// Mitsubishi GX Works2 project: RecipeMixer2   PLC: FX3U/FX3UC

PROGRAM MAIN
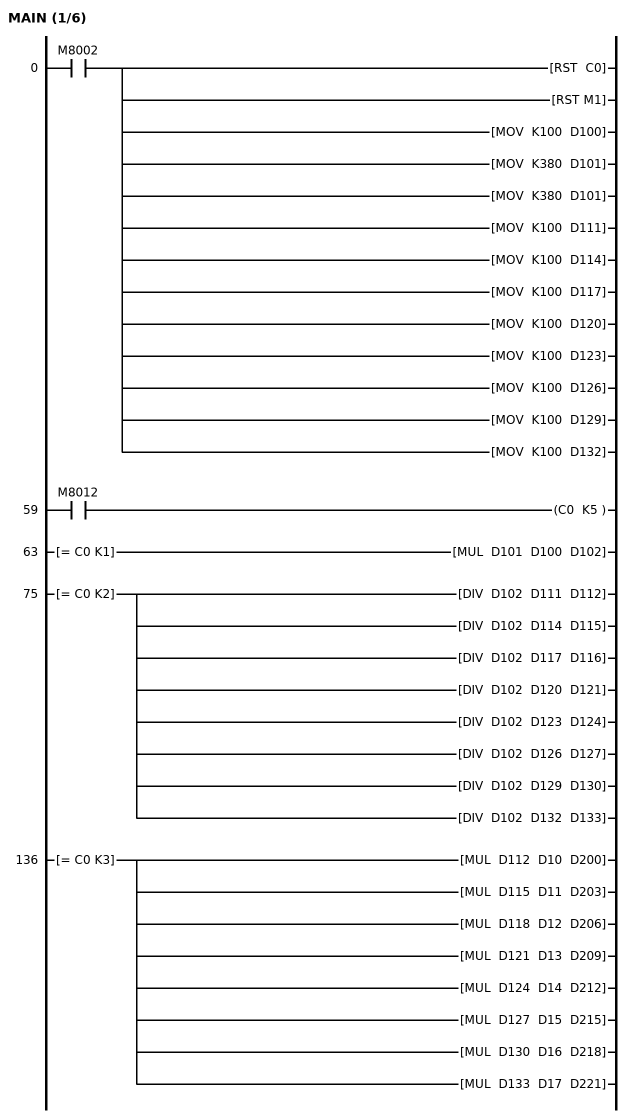
0     LD      M8002
      RST     C0
      RST     M1
      MOV     K100 D100
      MOV     K380 D101
      MOV     K380 D101
      MOV     K100 D111
      MOV     K100 D114
      MOV     K100 D117
      MOV     K100 D120
      MOV     K100 D123
      MOV     K100 D126
      MOV     K100 D129
      MOV     K100 D132
59    LD      M8012
      OUT     C0 K5
63    LD=     C0 K1
      MUL     D101 D100 D102
75    LD=     C0 K2
      DIV     D102 D111 D112
      DIV     D102 D114 D115
      DIV     D102 D117 D116
      DIV     D102 D120 D121
      DIV     D102 D123 D124
      DIV     D102 D126 D127
      DIV     D102 D129 D130
      DIV     D102 D132 D133
136   LD=     C0 K3
      MUL     D112 D10 D200
      MUL     D115 D11 D203
      MUL     D118 D12 D206
      MUL     D121 D13 D209
      MUL     D124 D14 D212
      MUL     D127 D15 D215
      MUL     D130 D16 D218
      MUL     D133 D17 D221
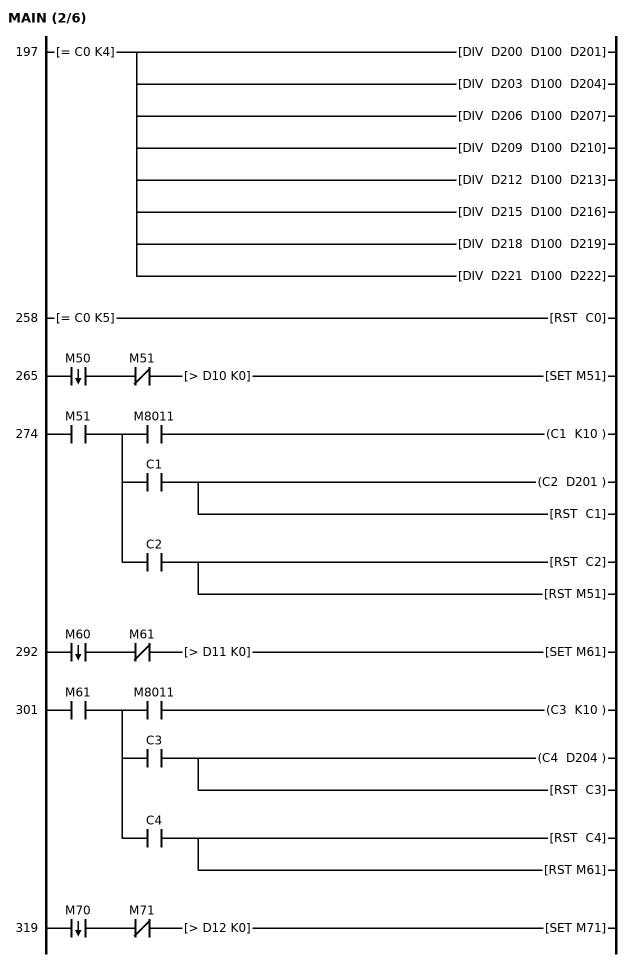
197   LD=     C0 K4
      DIV     D200 D100 D201
      DIV     D203 D100 D204
      DIV     D206 D100 D207
      DIV     D209 D100 D210
      DIV     D212 D100 D213
      DIV     D215 D100 D216
      DIV     D218 D100 D219
      DIV     D221 D100 D222
258   LD=     C0 K5
      RST     C0
265   LDF     M50
      ANI     M51
      AND>    D10 K0
      SET     M51
274   LD      M51
      MPS
      AND     M8011
      OUT     C1 K10
      MRD
      AND     C1
      OUT     C2 D201
      RST     C1
      MPP
      AND     C2
      RST     C2
      RST     M51
292   LDF     M60
      ANI     M61
      AND>    D11 K0
      SET     M61
301   LD      M61
      MPS
      AND     M8011
      OUT     C3 K10
      MRD
      AND     C3
      OUT     C4 D204
      RST     C3
      MPP
      AND     C4
      RST     C4
      RST     M61
319   LDF     M70
      ANI     M71
      AND>    D12 K0
      SET     M71
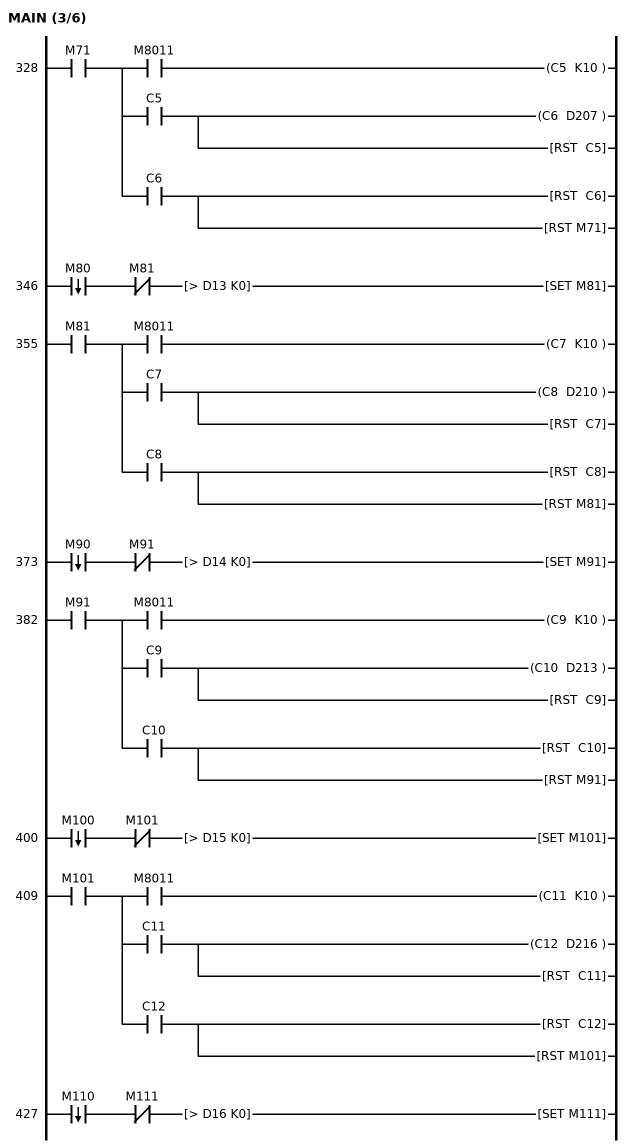
328   LD      M71
      MPS
      AND     M8011
      OUT     C5 K10
      MRD
      AND     C5
      OUT     C6 D207
      RST     C5
      MPP
      AND     C6
      RST     C6
      RST     M71
346   LDF     M80
      ANI     M81
      AND>    D13 K0
      SET     M81
355   LD      M81
      MPS
      AND     M8011
      OUT     C7 K10
      MRD
      AND     C7
      OUT     C8 D210
      RST     C7
      MPP
      AND     C8
      RST     C8
      RST     M81
373   LDF     M90
      ANI     M91
      AND>    D14 K0
      SET     M91
382   LD      M91
      MPS
      AND     M8011
      OUT     C9 K10
      MRD
      AND     C9
      OUT     C10 D213
      RST     C9
      MPP
      AND     C10
      RST     C10
      RST     M91
400   LDF     M100
      ANI     M101
      AND>    D15 K0
      SET     M101
409   LD      M101
      MPS
      AND     M8011
      OUT     C11 K10
      MRD
      AND     C11
      OUT     C12 D216
      RST     C11
      MPP
      AND     C12
      RST     C12
      RST     M101
427   LDF     M110
      ANI     M111
      AND>    D16 K0
      SET     M111
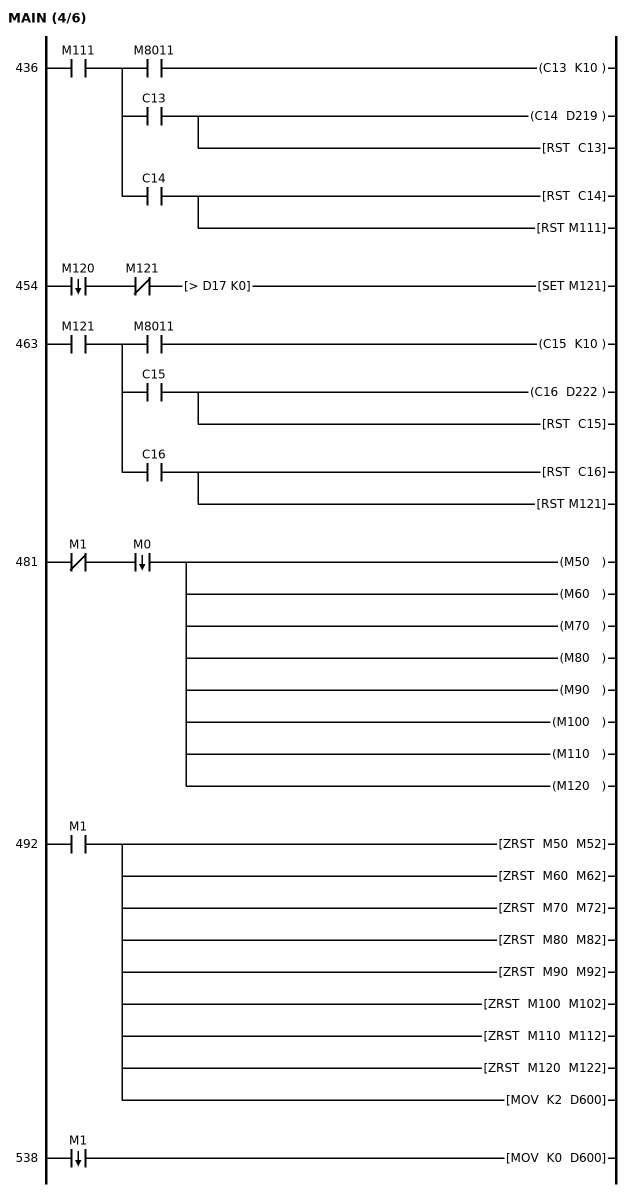
436   LD      M111
      MPS
      AND     M8011
      OUT     C13 K10
      MRD
      AND     C13
      OUT     C14 D219
      RST     C13
      MPP
      AND     C14
      RST     C14
      RST     M111
454   LDF     M120
      ANI     M121
      AND>    D17 K0
      SET     M121
463   LD      M121
      MPS
      AND     M8011
      OUT     C15 K10
      MRD
      AND     C15
      OUT     C16 D222
      RST     C15
      MPP
      AND     C16
      RST     C16
      RST     M121
481   LDI     M1
      ANDF    M0
      OUT     M50
      OUT     M60
      OUT     M70
      OUT     M80
      OUT     M90
      OUT     M100
      OUT     M110
      OUT     M120
492   LD      M1
      ZRST    M50 M52
      ZRST    M60 M62
      ZRST    M70 M72
      ZRST    M80 M82
      ZRST    M90 M92
      ZRST    M100 M102
      ZRST    M110 M112
      ZRST    M120 M122
      MOV     K2 D600
538   LDF     M1
      MOV     K0 D600
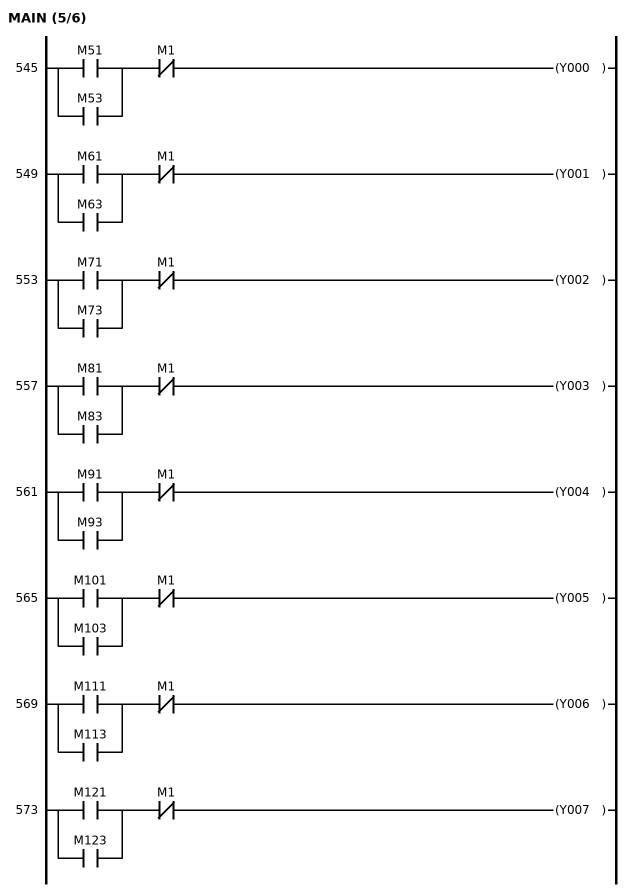
545   LD      M51
      OR      M53
      ANI     M1
      OUT     Y000
549   LD      M61
      OR      M63
      ANI     M1
      OUT     Y001
553   LD      M71
      OR      M73
      ANI     M1
      OUT     Y002
557   LD      M81
      OR      M83
      ANI     M1
      OUT     Y003
561   LD      M91
      OR      M93
      ANI     M1
      OUT     Y004
565   LD      M101
      OR      M103
      ANI     M1
      OUT     Y005
569   LD      M111
      OR      M113
      ANI     M1
      OUT     Y006
573   LD      M121
      OR      M123
      ANI     M1
      OUT     Y007
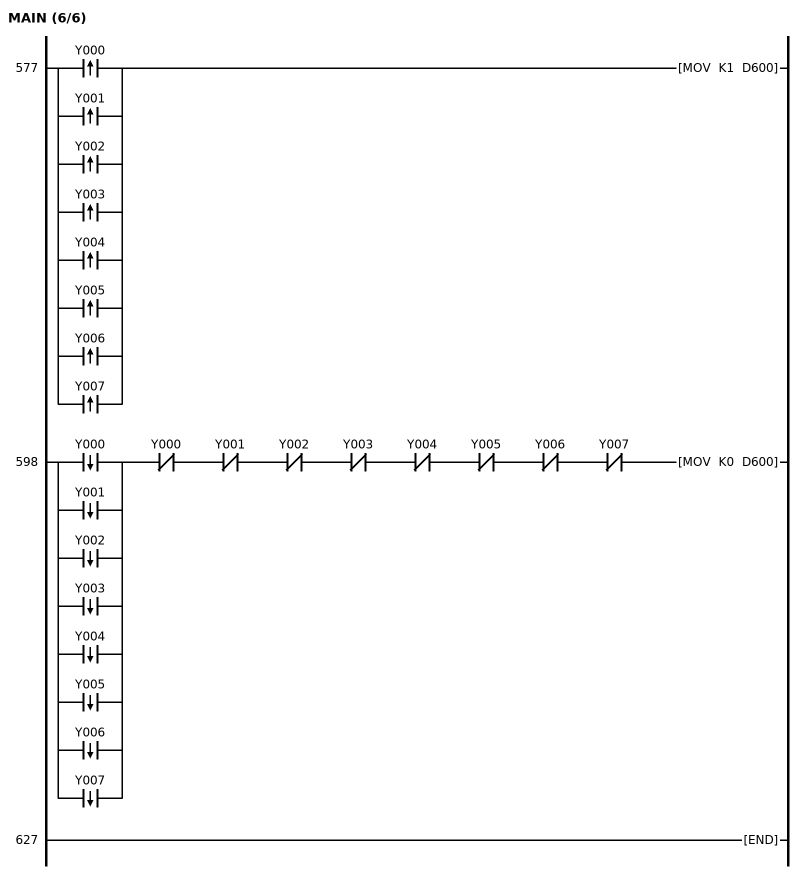
577   LDP     Y000
      ORP     Y001
      ORP     Y002
      ORP     Y003
      ORP     Y004
      ORP     Y005
      ORP     Y006
      ORP     Y007
      MOV     K1 D600
598   LDF     Y000
      ORF     Y001
      ORF     Y002
      ORF     Y003
      ORF     Y004
      ORF     Y005
      ORF     Y006
      ORF     Y007
      ANI     Y000
      ANI     Y001
      ANI     Y002
      ANI     Y003
      ANI     Y004
      ANI     Y005
      ANI     Y006
      ANI     Y007
      MOV     K0 D600
627   END
END_PROGRAM
